SUBAPPLICATION Uebung_102 (* DigitalInput_I1/I2 auf DigitalOutput_Q1, mit Plug and Socket *)
  (* Standard: 61499-2; Description: Copyright (c) 2023 Meisterschulen am Ostbahnhof This program and the accompanying materials are made available under the terms of the Eclipse Public License 2.0 which is available at https://www.eclipse.org/legal/epl-2.0/ SPDX-License-Identifier: EPL-2.0 *)
  (* Version 1.0, 2023-10-23, Franz Höpfinger, Meisterschulen am Ostbahnhof *)
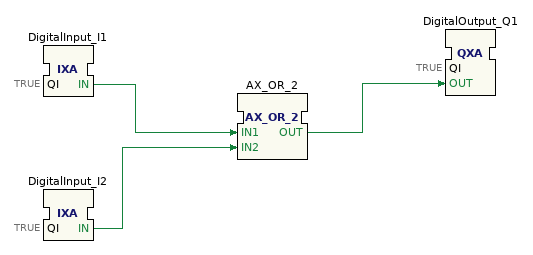
  FBS
    DigitalInput_I1 : IXA(QI := TRUE);
    DigitalOutput_Q1 : QXA(QI := TRUE);
    AX_OR_2 : AX_OR_2;
    DigitalInput_I2 : IXA(QI := TRUE);
  END_FBS
  ADAPTER_CONNECTIONS
    AX_OR_2.OUT TO DigitalOutput_Q1.OUT;
    DigitalInput_I1.IN TO AX_OR_2.IN1;
    DigitalInput_I2.IN TO AX_OR_2.IN2;
  END_CONNECTIONS
END_SUBAPPLICATION
